FUNCTION alg_a_pusher3 : BOOL
VAR_INPUT
	state: STATE;
END_VAR

alg_a_pusher3 := FALSE;

END_FUNCTION

(* stored: Version 1.1.0.1, ProductVersion 3.1.4022.18
   POU alg_a_pusher3: Id {c9772f25-8ced-45fd-a76e-96a37fa31c84}, SpecialFunc None *)
